PROGRAM PRG_01_Reel
VAR
END_VAR

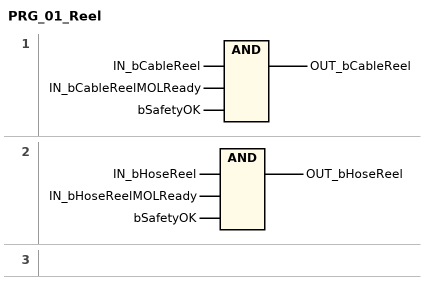
// NETWORK 1
OUT_bCableReel := IN_bCableReel AND IN_bCableReelMOLReady AND bSafetyOK;

// NETWORK 2
OUT_bHoseReel := IN_bHoseReel AND IN_bHoseReelMOLReady AND bSafetyOK;

// NETWORK 3

END_PROGRAM

(* stored: Version 1.1.0.1, ProductVersion 3.1.4024.12
   POU PRG_01_Reel: Id {331bba7a-39ea-4280-a069-5c09484cbbbc}, SpecialFunc None *)
